INTERFACE ITcoDialogFormat

METHOD WithCaption : ITcoDialogAnswer
VAR_INPUT
	inCaption : STRING(255);
END_VAR
END_METHOD

METHOD WithOk : ITcoDialogAnswer
VAR_INPUT
END_VAR
END_METHOD

METHOD WithText : ITcoDialogAnswer
VAR_INPUT
	inText : STRING(500);
END_VAR
END_METHOD

METHOD WithYesNo : ITcoDialogAnswer
VAR_INPUT
END_VAR
END_METHOD

METHOD WithYesNoCancel : ITcoDialogAnswer
END_METHOD

END_INTERFACE

(* stored: Version 1.1.0.1
   Itf ITcoDialogFormat: Id {c2d6a20f-376b-0b37-309b-4fbaea25ba73}
   Folder Format: Id {ef2bd4fc-2ef1-02f5-28b3-bdea702f0ebe}
   Method WithCaption: Id {256464fc-5542-0c19-1dbe-d5ab79664f30}
   Method WithOk: Id {e2f96920-7b83-023e-28d1-33a200d8eadf}
   Method WithText: Id {0aefd627-5574-002d-1f07-a884440c512d}
   Method WithYesNo: Id {65f97506-e622-06fa-3050-66f1ebb81bab}
   Method WithYesNoCancel: Id {64016aeb-0530-0115-02e5-e4e68fe22a83} *)
